FUNCTION F_GetOrientationST : BOOL
VAR_INPUT
	SrcContour		: ITcVnContainer;
    ipDestImage : Reference To  ITcVnImage;
    eTransform  : ETcVnColorSpaceTransform;
    hrPrev      : HRESULT;
END_VAR
VAR
	size : ULINT;
END_VAR

size := SrcContour.GetElementNum;
//getElementNum is # of elements
//getElementSize is byte size
for

END_FUNCTION

(* stored: Version 1.1.0.1, ProductVersion 3.1.4024.12
   POU F_GetOrientationST: Id {b2a17eef-20b7-4953-af58-15c2e2d33448}, SpecialFunc None *)
